// TIA Portal V14 SP1 program export: 0 tag tables, 0 data types, 0 data blocks, 1 code blocks (in call order from the OBs), 0 instance data blocks

ORGANIZATION_BLOCK "Main"   // OB1, LAD, ProgramCycle
TITLE = "Main Program Sweep (Cycle)"
{ S7_Optimized_Access := 'TRUE' }
VERSION : 0.1
// stored: AutoNumber true, CodeModifiedDate 2019-01-22T16:31:49.5601666Z, CompileDate 2019-01-22T16:31:55.0384488Z, CreationDate 2019-01-18T20:48:30.3502008Z, HandleErrorsWithinBlock false, InterfaceModifiedDate 2008-07-21T16:55:08.419547Z, IsConsistent true, IsIECCheckEnabled false, IsKnowHowProtected false, IsWriteProtected false, ModifiedDate 2019-01-22T16:33:48.3121731Z, ParameterModified 2008-07-21T16:55:08.419547Z, StructureModified 2008-07-21T16:55:08.419547Z
   VAR_INPUT
      Initial_Call : Bool;   // Initial call of this OB
      Remanence : Bool;   // =True, if remanent data are available
   END_VAR
   VAR_TEMP
      donewait : Bool;
      ntrig : Bool;
      triggerque : Bool;
      triggerque4 : Bool;
      errorrfid : Bool;
      status : DWord;
   END_VAR
BEGIN

REGION Network 1: conveyor
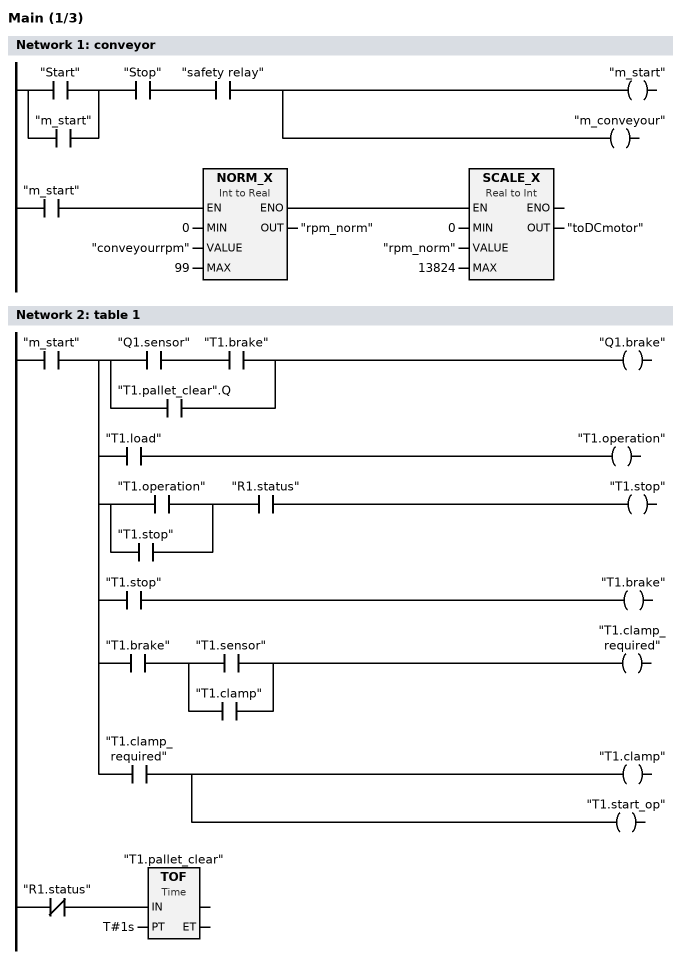
   RUNG wire#powerrail
      Contact( "Start" )
      wire#w1
      Contact( "Stop" )
      Contact( "safety relay" )
      wire#w2
      Coil( "m_start" )
   END_RUNG
   RUNG wire#powerrail
      Contact( "m_start" )
   END_RUNG wire#w1
   RUNG wire#w2
      Coil( "m_conveyour" )
   END_RUNG
   RUNG wire#powerrail
      Contact( "m_start" )
      { S7_Templates := "[SrcType := Int, DestType := Real]" } Normalize(min := 0, value := "conveyourrpm", max := 99, out => "rpm_norm")
      { S7_Templates := "[SrcType := Real, DestType := Int]" } Scale(min := 0, value := "rpm_norm", max := 13824, out => "toDCmotor")
   END_RUNG
   // the same network as SCL:
   "m_start" := ("Start" OR "m_start") AND "Stop" AND "safety relay";
   "m_conveyour" := "m_start";
   IF "m_start" THEN
       "rpm_norm" := NORM_X(MIN := 0, VALUE := "conveyourrpm", MAX := 99);
       "toDCmotor" := SCALE_X(MIN := 0, VALUE := "rpm_norm", MAX := 13824);
   END_IF;
END_REGION

REGION Network 2: table 1
   RUNG wire#powerrail
      Contact( "m_start" )
      wire#w1
      Contact( "Q1.sensor" )
      Contact( "T1.brake" )
      wire#w2
      Coil( "Q1.brake" )
   END_RUNG
   RUNG wire#w1
      Contact( "T1.pallet_clear".Q )
   END_RUNG wire#w2
   RUNG wire#w1
      Contact( "T1.load" )
      Coil( "T1.operation" )
   END_RUNG
   RUNG wire#w1
      Contact( "T1.operation" )
      wire#w3
      Contact( "R1.status" )
      Coil( "T1.stop" )
   END_RUNG
   RUNG wire#w1
      Contact( "T1.stop" )
   END_RUNG wire#w3
   RUNG wire#w1
      Contact( "T1.stop" )
      Coil( "T1.brake" )
   END_RUNG
   RUNG wire#w1
      Contact( "T1.brake" )
      wire#w4
      Contact( "T1.sensor" )
      wire#w5
      Coil( "T1.clamp_required" )
   END_RUNG
   RUNG wire#w4
      Contact( "T1.clamp" )
   END_RUNG wire#w5
   RUNG wire#w1
      Contact( "T1.clamp_required" )
      wire#w6
      Coil( "T1.clamp" )
   END_RUNG
   RUNG wire#w6
      Coil( "T1.start_op" )
   END_RUNG
   RUNG wire#powerrail
      I_Contact( "R1.status" )
      { S7_Templates := "time_type := Time" } "T1.pallet_clear".TOF(pt := T#1s, et =>)
   END_RUNG
   // the same network as SCL:
   "Q1.brake" := "m_start" AND (("Q1.sensor" AND "T1.brake") OR "T1.pallet_clear".Q);
   "T1.operation" := "m_start" AND "T1.load";
   "T1.stop" := "m_start" AND ("T1.operation" OR "T1.stop") AND "R1.status";
   "T1.brake" := "m_start" AND "T1.stop";
   "T1.clamp_required" := "m_start" AND "T1.brake" AND ("T1.sensor" OR "T1.clamp");
   "T1.clamp" := "m_start" AND "T1.clamp_required";
   "T1.start_op" := "T1.clamp";
   "T1.pallet_clear".TOF(IN := NOT "R1.status", PT := T#1s);
END_REGION

REGION Network 3: table 2
END_REGION

REGION Network 4: table 3
END_REGION

REGION Network 5: table 4
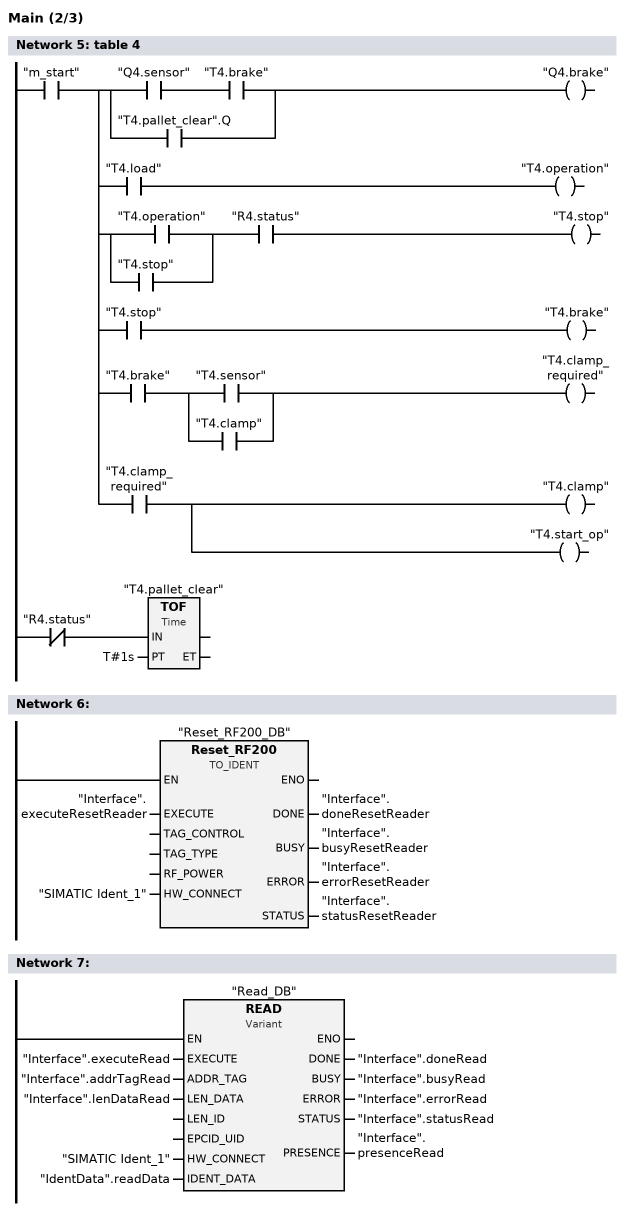
   RUNG wire#powerrail
      Contact( "m_start" )
      wire#w1
      Contact( "Q4.sensor" )
      Contact( "T4.brake" )
      wire#w2
      Coil( "Q4.brake" )
   END_RUNG
   RUNG wire#w1
      Contact( "T4.pallet_clear".Q )
   END_RUNG wire#w2
   RUNG wire#w1
      Contact( "T4.load" )
      Coil( "T4.operation" )
   END_RUNG
   RUNG wire#w1
      Contact( "T4.operation" )
      wire#w3
      Contact( "R4.status" )
      Coil( "T4.stop" )
   END_RUNG
   RUNG wire#w1
      Contact( "T4.stop" )
   END_RUNG wire#w3
   RUNG wire#w1
      Contact( "T4.stop" )
      Coil( "T4.brake" )
   END_RUNG
   RUNG wire#w1
      Contact( "T4.brake" )
      wire#w4
      Contact( "T4.sensor" )
      wire#w5
      Coil( "T4.clamp_required" )
   END_RUNG
   RUNG wire#w4
      Contact( "T4.clamp" )
   END_RUNG wire#w5
   RUNG wire#w1
      Contact( "T4.clamp_required" )
      wire#w6
      Coil( "T4.clamp" )
   END_RUNG
   RUNG wire#w6
      Coil( "T4.start_op" )
   END_RUNG
   RUNG wire#powerrail
      I_Contact( "R4.status" )
      { S7_Templates := "time_type := Time" } "T4.pallet_clear".TOF(pt := T#1s, et =>)
   END_RUNG
   // the same network as SCL:
   "Q4.brake" := "m_start" AND (("Q4.sensor" AND "T4.brake") OR "T4.pallet_clear".Q);
   "T4.operation" := "m_start" AND "T4.load";
   "T4.stop" := "m_start" AND ("T4.operation" OR "T4.stop") AND "R4.status";
   "T4.brake" := "m_start" AND "T4.stop";
   "T4.clamp_required" := "m_start" AND "T4.brake" AND ("T4.sensor" OR "T4.clamp");
   "T4.clamp" := "m_start" AND "T4.clamp_required";
   "T4.start_op" := "T4.clamp";
   "T4.pallet_clear".TOF(IN := NOT "R4.status", PT := T#1s);
END_REGION

REGION Network 6
   RUNG wire#powerrail
      { S7_Templates := "connect_type := TO_IDENT" } "Reset_RF200_DB".Reset_RF200(EXECUTE := "Interface".executeResetReader, TAG_CONTROL :=, TAG_TYPE :=, RF_POWER :=, HW_CONNECT := "SIMATIC Ident_1", DONE => "Interface".doneResetReader, BUSY => "Interface".busyResetReader, ERROR => "Interface".errorResetReader, STATUS => "Interface".statusResetReader)
   END_RUNG
   // the same network as SCL:
   "Reset_RF200_DB"(EXECUTE := "Interface".executeResetReader,   // Reset_RF200
                    HW_CONNECT := "SIMATIC Ident_1",
                    DONE => "Interface".doneResetReader,
                    BUSY => "Interface".busyResetReader,
                    ERROR => "Interface".errorResetReader,
                    STATUS => "Interface".statusResetReader);
END_REGION

REGION Network 7
   RUNG wire#powerrail
      { S7_Templates := "[ident_data_type := Variant, connect_type := TO_IDENT]" } "Read_DB".Read(EXECUTE := "Interface".executeRead, ADDR_TAG := "Interface".addrTagRead, LEN_DATA := "Interface".lenDataRead, LEN_ID :=, EPCID_UID :=, HW_CONNECT := "SIMATIC Ident_1", IDENT_DATA := "IdentData".readData, DONE => "Interface".doneRead, BUSY => "Interface".busyRead, ERROR => "Interface".errorRead, STATUS => "Interface".statusRead, PRESENCE => "Interface".presenceRead)
   END_RUNG
   // the same network as SCL:
   "Read_DB"(EXECUTE := "Interface".executeRead,   // Read
             ADDR_TAG := "Interface".addrTagRead,
             LEN_DATA := "Interface".lenDataRead,
             HW_CONNECT := "SIMATIC Ident_1",
             IDENT_DATA := "IdentData".readData,
             DONE => "Interface".doneRead,
             BUSY => "Interface".busyRead,
             ERROR => "Interface".errorRead,
             STATUS => "Interface".statusRead,
             PRESENCE => "Interface".presenceRead);
END_REGION

REGION Network 8
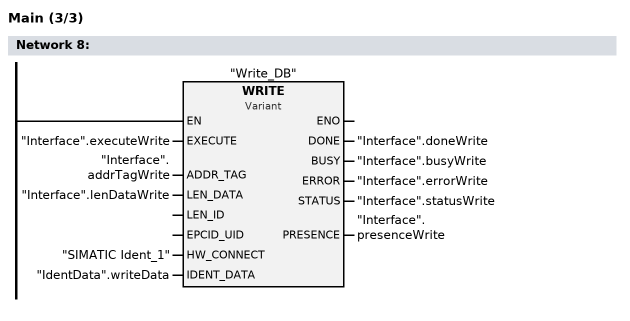
   RUNG wire#powerrail
      { S7_Templates := "[ident_data_type := Variant, connect_type := TO_IDENT]" } "Write_DB".Write(EXECUTE := "Interface".executeWrite, ADDR_TAG := "Interface".addrTagWrite, LEN_DATA := "Interface".lenDataWrite, LEN_ID :=, EPCID_UID :=, HW_CONNECT := "SIMATIC Ident_1", IDENT_DATA := "IdentData".writeData, DONE => "Interface".doneWrite, BUSY => "Interface".busyWrite, ERROR => "Interface".errorWrite, STATUS => "Interface".statusWrite, PRESENCE => "Interface".presenceWrite)
   END_RUNG
   // the same network as SCL:
   "Write_DB"(EXECUTE := "Interface".executeWrite,   // Write
              ADDR_TAG := "Interface".addrTagWrite,
              LEN_DATA := "Interface".lenDataWrite,
              HW_CONNECT := "SIMATIC Ident_1",
              IDENT_DATA := "IdentData".writeData,
              DONE => "Interface".doneWrite,
              BUSY => "Interface".busyWrite,
              ERROR => "Interface".errorWrite,
              STATUS => "Interface".statusWrite,
              PRESENCE => "Interface".presenceWrite);
END_REGION
END_ORGANIZATION_BLOCK
